// TIA Portal V16 export
// export: Created 2022-09-01T13:58:49.9529818Z, ExportSetting WithDefaults, DisplayName Totally Integrated Automation Portal, DisplayVersion V16, DisplayName TIA Portal Version Control Interface, DisplayVersion V16, DisplayName TIA Portal Openness, DisplayVersion V16, DisplayName STEP 7 Professional, DisplayVersion V16, DisplayName STEP 7 Safety, DisplayVersion V16, DisplayName WinCC Advanced, DisplayVersion V16
ORGANIZATION_BLOCK "Main"   // OB1, LAD, ProgramCycle
TITLE = "Main Program Sweep (Cycle)"
{ S7_Optimized_Access := 'TRUE' }
VERSION : 0.1
// stored: AutoNumber true, IsIECCheckEnabled false, SetENOAutomatically false
   VAR_INPUT
      Initial_Call : Bool;   // Initial call of this OB
      Remanence : Bool;   // =True, if remanent data are available
   END_VAR
   VAR_TEMP   // added for the SCL form of the ladder/FBD networks
      _w1 : Bool;
   END_VAR
BEGIN

REGION Network 1: Ciclo de lavagem e enxaguamento
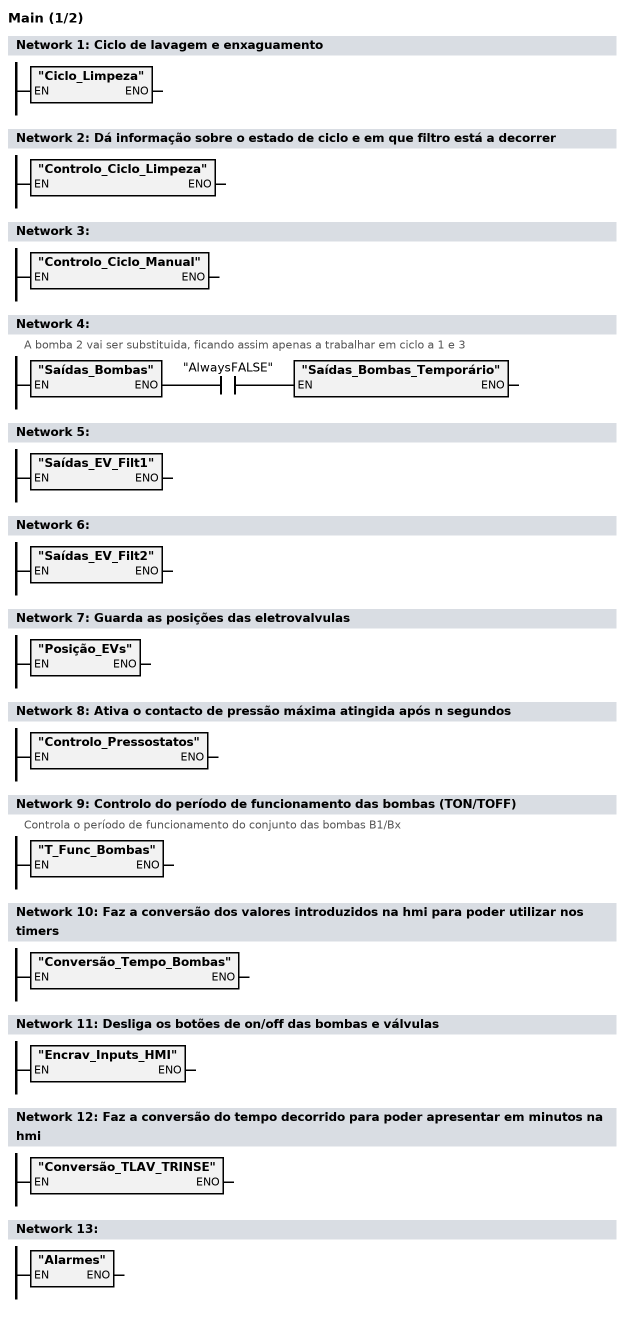
   RUNG wire#powerrail
      "Ciclo_Limpeza"()
   END_RUNG
   // the same network as SCL:
   "Ciclo_Limpeza"();
END_REGION

REGION Network 2: Dá informação sobre o estado de ciclo e em que filtro está a decorrer
   RUNG wire#powerrail
      "Controlo_Ciclo_Limpeza"()
   END_RUNG
   // the same network as SCL:
   "Controlo_Ciclo_Limpeza"();
END_REGION

REGION Network 3
   RUNG wire#powerrail
      "Controlo_Ciclo_Manual"()
   END_RUNG
   // the same network as SCL:
   "Controlo_Ciclo_Manual"();
END_REGION

REGION Network 4
   // A bomba 2 vai ser substituida, ficando assim apenas a trabalhar em ciclo a 1 e 3
   RUNG wire#powerrail
      "Saídas_Bombas"()
      Contact( "AlwaysFALSE" )
      "Saídas_Bombas_Temporário"()
   END_RUNG
   // the same network as SCL:
   "Saídas_Bombas"(ENO => #_w1);
   IF #_w1 AND "AlwaysFALSE" THEN "Saídas_Bombas_Temporário"(); END_IF;
END_REGION

REGION Network 5
   RUNG wire#powerrail
      "Saídas_EV_Filt1"()
   END_RUNG
   // the same network as SCL:
   "Saídas_EV_Filt1"();
END_REGION

REGION Network 6
   RUNG wire#powerrail
      "Saídas_EV_Filt2"()
   END_RUNG
   // the same network as SCL:
   "Saídas_EV_Filt2"();
END_REGION

REGION Network 7: Guarda as posições das eletrovalvulas
   RUNG wire#powerrail
      "Posição_EVs"()
   END_RUNG
   // the same network as SCL:
   "Posição_EVs"();
END_REGION

REGION Network 8: Ativa o contacto de pressão máxima atingida após n segundos
   RUNG wire#powerrail
      "Controlo_Pressostatos"()
   END_RUNG
   // the same network as SCL:
   "Controlo_Pressostatos"();
END_REGION

REGION Network 9: Controlo do período de funcionamento das bombas (TON/TOFF)
   // Controla o período de funcionamento do conjunto das bombas B1/Bx
   RUNG wire#powerrail
      "T_Func_Bombas"()
   END_RUNG
   // the same network as SCL:
   "T_Func_Bombas"();
END_REGION

REGION Network 10: Faz a conversão dos valores introduzidos na hmi para poder utilizar nos timers
   RUNG wire#powerrail
      "Conversão_Tempo_Bombas"()
   END_RUNG
   // the same network as SCL:
   "Conversão_Tempo_Bombas"();
END_REGION

REGION Network 11: Desliga os botões de on/off das bombas e válvulas
   RUNG wire#powerrail
      "Encrav_Inputs_HMI"()
   END_RUNG
   // the same network as SCL:
   "Encrav_Inputs_HMI"();
END_REGION

REGION Network 12: Faz a conversão do tempo decorrido para poder apresentar em minutos na hmi
   RUNG wire#powerrail
      "Conversão_TLAV_TRINSE"()
   END_RUNG
   // the same network as SCL:
   "Conversão_TLAV_TRINSE"();
END_REGION

REGION Network 13
   RUNG wire#powerrail
      "Alarmes"()
   END_RUNG
   // the same network as SCL:
   "Alarmes"();
END_REGION

REGION Network 14: Ultravioleta
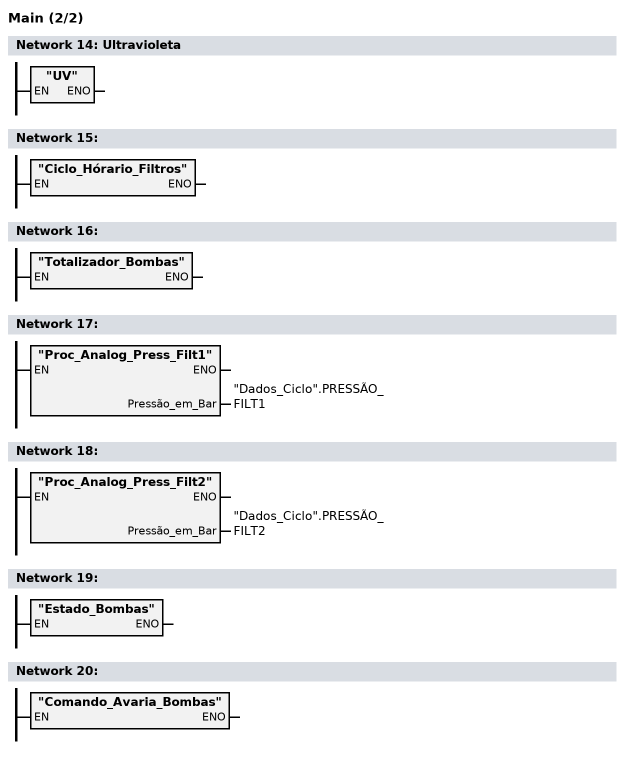
   RUNG wire#powerrail
      "UV"()
   END_RUNG
   // the same network as SCL:
   "UV"();
END_REGION

REGION Network 15
   RUNG wire#powerrail
      "Ciclo_Hórario_Filtros"()
   END_RUNG
   // the same network as SCL:
   "Ciclo_Hórario_Filtros"();
END_REGION

REGION Network 16
   RUNG wire#powerrail
      "Totalizador_Bombas"()
   END_RUNG
   // the same network as SCL:
   "Totalizador_Bombas"();
END_REGION

REGION Network 17
   RUNG wire#powerrail
      "Proc_Analog_Press_Filt1"(Pressão_em_Bar => "Dados_Ciclo".PRESSÃO_FILT1)
   END_RUNG
   // the same network as SCL:
   "Proc_Analog_Press_Filt1"(Pressão_em_Bar => "Dados_Ciclo".PRESSÃO_FILT1);
END_REGION

REGION Network 18
   RUNG wire#powerrail
      "Proc_Analog_Press_Filt2"(Pressão_em_Bar => "Dados_Ciclo".PRESSÃO_FILT2)
   END_RUNG
   // the same network as SCL:
   "Proc_Analog_Press_Filt2"(Pressão_em_Bar => "Dados_Ciclo".PRESSÃO_FILT2);
END_REGION

REGION Network 19
   RUNG wire#powerrail
      "Estado_Bombas"()
   END_RUNG
   // the same network as SCL:
   "Estado_Bombas"();
END_REGION

REGION Network 20
   RUNG wire#powerrail
      "Comando_Avaria_Bombas"()
   END_RUNG
   // the same network as SCL:
   "Comando_Avaria_Bombas"();
END_REGION
END_ORGANIZATION_BLOCK
